	            // Direction error
	            IF #sUDT_HMIStatus.Specific.DirectionErr                                  // Direction verification found the direction fault, stop VSU action and move in opposite direction
	                AND NOT #iqUDT_VSUInterface.MotorRunning                               // The VFD is stopped
	                AND #sx_PEC_EoSFiltered                                                 // The photoeye on the VSU conveyor is empty
	            THEN

	                #sUDT_HMIStatus.Specific.DirectionErr := FALSE;                       // Direction verification found the direction fault, stop VSU action and move in opposite direction

	            END_IF;

	        END_IF;
	    END_REGION

	    REGION 2.2 - Set errors

	        // Exit gap check blocked in movement
	        IF NOT #sx_PEC_GapEnd                                                             // Upper jam sensor occupied
	            AND #iqUDT_VSUInterface.Positioning                                        // The positioning motor is running
	            AND (#sx_UpRequest OR #sx_DownRequest)                                                         // an uprequest is active (going up)
	        THEN

	            #sUDT_HMIStatus.Specific.ExitGapErr := TRUE;                      // Set error upper jam sensor
	        END_IF;

	        // Entry gap check blocked in movement
	        IF NOT #sx_PEC_GapBegin                                                           // Lower jam sensor occupied
	            AND #iqUDT_VSUInterface.Positioning                                        // The positioning motor is running
	            AND (#sx_UpRequest OR #sx_DownRequest)                                                       // an downrequest is active (going down)
	        THEN

	            #sUDT_HMIStatus.Specific.EntryGapErr := TRUE;                      // Set error lower jam sensor
	        END_IF;


	        // Belt tear switch 1
	        IF NOT #ix_BeltTear1                                                   // Belt tear switch 1 is activated
	        THEN
	            #sUDT_HMIStatus.Specific.BeltTear1Err := TRUE;                // set error
	        END_IF;

	        // Belt tear switch 2
	        IF NOT #ix_BeltTear2                                                   // Belt tear switch 2 is activated
	        THEN
	            #sUDT_HMIStatus.Specific.BeltTear2Err := TRUE;                // set error
	        END_IF;

	        // Maintenace supports for lift carriage extracted
	        IF NOT #ix_MaintSupport1                                               // Maintenace support 1 extended
	        THEN
	            #sUDT_HMIStatus.Specific.MaintSupport1Err := TRUE;             // set error
	        END_IF;

	        // Maintenace supports for lift carriage extracted
	        IF NOT #ix_MaintSupport2                                                // Maintenace support 2 extended
	        THEN
	            #sUDT_HMIStatus.Specific.MaintSupport2Err := TRUE;             // set error
	        END_IF;

	        // Upper limit switch
	        IF #ix_LimitSwitchUp                                                   // Upper limit switch is overrun
	        THEN
	            #sUDT_HMIStatus.Specific.UpperPositionErr := TRUE;             // set error
	        END_IF;

	        IF NOT #ix_SafetyDoorDiagUp                                                 // Safety door diagnostic output
	        THEN
	            #sUDT_HMIStatus.Specific.SafetyDoorUpErr := TRUE;                // set error
	        END_IF;


	        // Lower limit switch
	        IF #ix_LimitSwitchDown                                                // Lower limit switch is overrun
	        THEN
	            #sUDT_HMIStatus.Specific.LowerPositionErr := TRUE;            // set error
	        END_IF;

	        IF NOT #ix_SafetyDoorDiagDown                                                 // Safety door diagnostic output
	        THEN
	            #sUDT_HMIStatus.Specific.SafetyDoorDownErr := TRUE;                // set error
	        END_IF;

	        // Direction fault in semiautomatic mode
	        IF #sx_SemiAutomatic                                                               // Running Semi-Automatic
	            AND (((#si_Position = #ci_PositionDown                                     // the requested position is "down"
	            AND #si_DefaultPosition = #ci_PositionDown)                                // and the configured "default" is equal to "down"
	            OR (#si_Position = #ci_PositionDefault                                     // or the request is "default"
	            AND #si_DefaultPosition = #ci_PositionDown)                                // and the configured "default" is equal to "down"
	            AND #sx_DownRequest)                                                       // but the position is "down"

	            OR ((#si_Position = #ci_PositionUp                                         // or the requested position is "up"
	            AND #si_DefaultPosition = #ci_PositionUp)                                  // and the configured "default" is equal to "up"
	            OR (#si_Position = #ci_PositionDefault                                     // or the request is "default"
	            AND #si_DefaultPosition = #ci_PositionUp)                                  // and the configured "default" is equal to "up"
	            AND #sx_UpRequest))                                                        // but the position is "up"
	        THEN

	            #sUDT_HMIStatus.Specific.DirectionErr := TRUE;                            // Direction verification found the Direction fault, stop the parcel
	        END_IF;



	        #sx_ConfigurationError := (#iUDT_VSUConfig.DefaultPosition <= 0);                  // Set the configuration error bit (No status!!)

	    END_REGION

	    REGION 2.3 - Common Error

	        #sUDT_Status.Error :=
	        #iqUDT_VSUInterface.InternalErrorVFD                                           // or there are errors in the VFD
	        OR #iqUDT_VSUInterface.InternalErrorRIOPanel                                   // or an internal error in the RIO panel occured
	        OR #sUDT_HMIStatus.Specific.DirectionErr                                      // Direction verification found the Direction fault, stop the parcel
	        OR #sUDT_HMIStatus.Specific.ExitGapErr                                // Upper jam PEC detected WHILE going Up
	        OR #sUDT_HMIStatus.Specific.EntryGapErr                                // Lower jam PEC detected while going Down
	        OR #sUDT_HMIStatus.Specific.MaintSupport1Err                            // Maintenace carriage support 1 extended in automatic mode
	        OR #sUDT_HMIStatus.Specific.MaintSupport2Err                            // Maintenace carriage support 2 extended in automatic mode
	        OR #sUDT_HMIStatus.Specific.BeltTear1Err                               // Belt tear sensor 1 was detected
	        OR #sUDT_HMIStatus.Specific.BeltTear2Err                              // Belt tear sensor 2 was detected
	        OR #sUDT_HMIStatus.Specific.UpperPositionErr                             // Upper limit switch is overrun
	        OR #sUDT_HMIStatus.Specific.LowerPositionErr                            // Lower limit switch is overrun
	        OR #sUDT_HMIStatus.Specific.SafetyDoorDownErr;                              // Safety door diagnostic fault

	    END_REGION

	    REGION 2.4 - Common Warning

	        // Keyswitch NOT in a position
	        #sUDT_HMIStatus.Specific.KeyswitchWrn := NOT #ix_LCPAutoMode AND NOT #ix_LCPManualMode;
	        #sUDT_Status.Warning := #sUDT_HMIStatus.Specific.KeyswitchWrn;

	    END_REGION

	END_REGION

	REGION 3 - Check conditions to set Equipment ready

	    //Conditions to set bit sx_Ready to operate

	    #sx_Ready := NOT #sUDT_Status.Error                                                // Error present
	    AND #ix_SafetyOk                                                                    // Safety signalling NOT OK
	    AND #iqUDT_VSUInterface.VSUMainPowerOk;                                             // 400v signalling not OK

	    //Enble main contactor
	    #qx_MainContactorOn := (#ix_LCPManualMode OR #ix_LCPAutoMode)                       // Auto or manual enabled
	    AND #ix_OverTempBrakingResistor;                                                    //Temperature breaking resistor is OK


	END_REGION

	REGION 4 - Stop Equipment

	    IF #sx_ManualModeActive                                                             // Manual mode is active
	        AND #sx_AutomaticActive

	        OR (NOT #iqUDT_EquipmentControl.Command.AutomaticOn                            // VSU stops if the bit AutomaticOn from control block is false
	        AND NOT #sx_ManualModeActive)                                                   // Manual mode active bit

	        OR (NOT #sx_Ready                                                               // Bit VSU ready to run in automatic mode
	        AND NOT #sx_ManualModeActive)                                                   // Manual mode active

	        OR NOT #ix_LCPAutoMode                                                          // LCP is not set to automatic
	        OR NOT #ix_SafetyOk                                                             //

	    THEN                                                                                // Order to stop
	        #sx_Stopping := TRUE;                                                           // stopping is activated
	        #sx_AutomaticActive := FALSE;                                                   // switch of automatic activ
	        #sx_StartReceived := FALSE;                                                     // Start command received from system

	    END_IF;

	    IF (#sx_Stopping                                                                     // stopping is activated
	        AND NOT #iqUDT_VSUInterface.Positioning)                                        // The positioning device is not active positioning
	        OR #sFB_MaxStopTime.qx_DelayedSignal
	        OR NOT #sx_Ready

	    THEN
	        #sx_Stopping := FALSE;                                                          // stopping is activated
	        #iqUDT_VSUCommand.CommandUp := FALSE;
	        #iqUDT_VSUCommand.CommandDown := FALSE;
	    END_IF;

	END_REGION

	REGION 5 - Start Automatic mode

	    REGION 5.1 - Start
	        // if start (OS) is received from system, this is memorised until started in cascade
	        IF #iqUDT_EquipmentControl.Command.Start                                       // Start from system
	            AND #sx_Ready                                                               // Equipment has no errors
	        THEN

	            #sx_StartReceived := TRUE;                                                  // Start command received from system

	        END_IF;

	        IF #sx_StartReceived                                                            // Start command received from system
	            AND #iqUDT_VSUInterface.Referenced                                         // and VSU is referenced
	            AND #ix_LCPAutoMode                                                         // and the LCP is set to auto
	        THEN

	            #sx_AutomaticActive := TRUE;                                                // Automatic activated
	            #sx_StartReceived := FALSE;                                                 // Start command received from system
	        END_IF;
	    END_REGION

	    REGION 5.2 - Semi automatic mode

	        #sx_SemiAutomatic := #sx_AutomaticActive                                        // Automatic activated
	        AND #iqUDT_VSUCommand.SemiAutomaticMode;                                       // and Semi-automatic is selected

	    END_REGION

	END_REGION

	REGION 6 - Manual mode

	    REGION 6.1 - Manual mode: activation

	        // Manual mode is active if it is active from hmi or by control block
	        #sx_ManualModeActive := #iqUDT_VSUCommand.ManualMode
	        OR #iqUDT_EquipmentControl.Command.ManualMode
	        OR #ix_LCPManualMode;

	    END_REGION

	    REGION 6.2 - Jog signals

	        #sx_CombinedJogUp :=
	        (((#iqUDT_VSUCommand.ManualMode                                                // HMI in manual
	        OR #iqUDT_EquipmentControl.Command.ManualMode)                                 // Or a system control command to go to manual
	        AND #iqUDT_VSUCommand.JogUp)                                                   // If selected jog in positive direction
	        OR (#ix_LCPManualMode                                                           // box in manual
	        AND #ix_LCPUp));                                                                // If selected jog in positive direction

	        #sx_CombinedJogDown :=
	        (((#iqUDT_VSUCommand.ManualMode                                                 // HMI in manual
	        OR #iqUDT_EquipmentControl.Command.ManualMode)                                  // Or a system control command to go to manual
	        AND #iqUDT_VSUCommand.JogDown)                                                 // If selected jog in negative direction
	        OR (#ix_LCPManualMode                                                           // box in manual
	        AND #ix_LCPDown));                                                              // If selected jog in negative direction

	        // Detecting rising edge on manual jog Up
	        #sR_TRIG_ManualJogUp(CLK := #sx_CombinedJogUp);

	        // Detecting rising edge on manual jog Down
	        #sR_TRIG_ManualJogDown(CLK := #sx_CombinedJogDown);

	    END_REGION

	    REGION 6.3 - Manual mode: disabled

	        // Manual mode bits inputs can be reset in case of malfunction
	        IF #iqUDT_EquipmentControl.Command.DisableManualMode
	        THEN

	            #iqUDT_VSUCommand.ManualMode := FALSE;                                     // reset manual mode
	            #iqUDT_EquipmentControl.Command.ManualMode := FALSE;                       // reset manual mode command
	            #iqUDT_VSUCommand.JogUp := FALSE;                                          // reset manual command Jog Up
	            #iqUDT_VSUCommand.JogDown := FALSE;                                        // reset manual command Jog Down
	            #sx_Jog := FALSE;
	        END_IF;
	    END_REGION

	    REGION 6.4 - Manual PreStart up or down

	        // Pre start conditions to run in manual mode
	        #sx_PreStartManual := #sx_ManualModeActive                                      // Manual mode active bit
	        AND #ix_SafetyOk                                                                // Safety healthy bit
	        //AND #iq_UDT_VSUInterface.PNDeviceOk                                                              // Profinet comunication
	        AND NOT #iqUDT_VSUInterface.InternalErrorVFD;                                  // Internal error from VFD

	        IF #sx_PreStartManual                                                           // Pre start conditions to run in manual mode
	            AND (#sR_TRIG_ManualJogUp.Q                                                  // Trigger to start VSU run in manual jog mode UP
	            OR #sR_TRIG_ManualJogDown.Q)                                                 // Trigger to start VSU run in manual jog mode Down
	            AND NOT #sFB_JogEnable.qx_DelayedSignal
	        THEN

	            #iqUDT_EquipmentControl.Request.SignalingRequest := TRUE;                  // Request signaling TO control block before VSU runs in manual mode

	        END_IF;

	    END_REGION

	    REGION 6.5 - Jog mode Up / Down

	        IF #sx_PreStartManual                                                           // IF in manual jog mode
	            AND (NOT #iqUDT_EquipmentControl.Request.SignalingRequest                  // Signaling request done
	            OR #sFB_JogEnable.qx_DelayedSignal)
	            AND #sx_CombinedJogUp                                                       // If selected jog in positive direction
	            AND NOT #sx_CombinedJogDown                                                 // And not selected jog in negative direction
	        THEN

	            #iqUDT_VSUInterface.JogUp := TRUE;                                         // set jog positive
	            #iqUDT_VSUInterface.JogDown := FALSE;                                      // reset jog negative
	            #sx_Jog := true;

	        ELSIF
	            #sx_PreStartManual                                                          // IF in manual jog mode
	            AND (NOT #iqUDT_EquipmentControl.Request.SignalingRequest                  // Signaling request done
	            OR #sFB_JogEnable.qx_DelayedSignal)
	            AND NOT #sx_CombinedJogUp                                                   // If selected jog in positive direction
	            AND #sx_CombinedJogDown                                                     // and there is command to jog in negative direction
	        THEN

	            #iqUDT_VSUInterface.JogUp := FALSE;                                        // reset jog positive
	            #iqUDT_VSUInterface.JogDown := TRUE;                                       // set jog negative
	            #sx_Jog := true;

	        ELSIF
	            NOT #sx_PreStartManual                                                      // If not in manual mode
	            OR (#sx_PreStartManual                                                      // or in manual mode
	            AND (#sx_CombinedJogUp                                                      // and jog positive is off
	            AND #sx_CombinedJogDown)                                                    // AND jog negative is off
	            OR (NOT #sx_CombinedJogUp                                                   // or jog positive is on
	            AND NOT #sx_CombinedJogDown))                                               // and jog negative is on
	        THEN

	            #iqUDT_VSUInterface.JogUp := FALSE;                                        // reset jog positive
	            #iqUDT_VSUInterface.JogDown := FALSE;                                      // reset jog negative
	            #sx_Jog := False;
	        END_IF;
	    END_REGION
	END_REGION

	REGION 7 - Automatic mode

	    REGION 7.1 - Direction from decision point
	        IF #iqUDT_VSUInterface.RequestedPosition <> 0                                  // Position is received from decision block
	        THEN
	            #si_Position := #iqUDT_VSUInterface.RequestedPosition;                     // Copy the input to the memory

	        END_IF;

	        // Requested position reset
	        IF (#iqUDT_VSUInterface.RequestedPosition = #iqUDT_VSUInterface.PositionActual OR
	            (#iqUDT_VSUInterface.RequestedPosition = #ci_PositionDefault AND #iqUDT_VSUInterface.PositionActual = #si_DefaultPosition))
	        THEN

	            #iqUDT_VSUInterface.RequestedPosition := 0;

	        END_IF;


	    END_REGION

	    REGION 7.2 - Position Up / Down
	        // 2 = Up, 1 = Down and 99 = Default
	        //
	        IF (#si_Position = #ci_PositionUp                                                            // If the position "up" is equal to the request
	            OR (#si_Position = #ci_PositionDefault                                                       // Or the request is "default"
	            AND #si_DefaultPosition = #ci_PositionUp))                                               // and the configured "default" is equal to "up"
	            AND #sx_Ready                                                               // Ready to operate, No errors active
	            AND #sx_AutomaticActive                                                     // Automaticly started
	            AND NOT #sx_SemiAutomatic                                                   // Not running Semi-Automatic
	        THEN

	            #sx_DownRequest := FALSE;                                                   // Reset down command
	            #sx_UpRequest := TRUE;                                                      // Set up command
	            #si_Position := 0;                                                          // Reset the memory
	        END_IF;

	        IF (#si_Position = #ci_PositionDown                                                            // If the position "down" is equal to the request
	            OR (#si_Position = #ci_PositionDefault                                                       // Or the request is "default"
	            AND #si_DefaultPosition = #ci_PositionDown))                                               // and the configured "default" is equal to "down"
	            AND #sx_Ready                                                               // Ready to operate, No errors active
	            AND #sx_AutomaticActive                                                     // Automaticly started
	            AND NOT #sx_SemiAutomatic                                                   // Not running Semi-Automatic
	        THEN

	            #sx_DownRequest := TRUE;                                                    // Set down command
	            #sx_UpRequest := FALSE;                                                     // Reset up command
	            #si_Position := 0;                                                          // Reset the memory
	        END_IF;

	        // if the VSU is not referenced set the default position, this ensures the VSU to go to the default
	        // after refferecing.

	        IF NOT #iqUDT_VSUInterface.Referenced
	        THEN
	            IF #si_DefaultPosition = #ci_PositionUp
	            THEN
	                #sx_DownRequest := FALSE;                                               // Reset down command
	                #sx_UpRequest := TRUE;                                                  // Set up command
	                #iqUDT_VSUInterface.PositionSetpoint := #ci_PositionUp;                             // Set position to be Up
	            END_IF;

	            IF #si_DefaultPosition = #ci_PositionDown
	            THEN
	                #sx_DownRequest := TRUE;                                                // Reset down command
	                #sx_UpRequest := FALSE;                                                 // Set up command
	                #iqUDT_VSUInterface.PositionSetpoint := #ci_PositionDown;                             // Set position to be Down
	            END_IF;
	        END_IF;

	    END_REGION

	    REGION 7.3 - Semi automatic

	        IF #sx_SemiAutomatic                                                            // Not running Semi-Automatic
	            AND #iqUDT_VSUCommand.CommandUp

	        THEN
	            #sx_DownRequest := FALSE;                                                   // Reset down command
	            #sx_UpRequest := TRUE;                                                      // Set up command
	            #iqUDT_VSUCommand.CommandUp := FALSE;
	        END_IF;

	        IF #sx_SemiAutomatic                                                            // Not running Semi-Automatic
	            AND #iqUDT_VSUCommand.CommandDown

	        THEN
	            #sx_DownRequest := TRUE;                                                    // Reset down command
	            #sx_UpRequest := FALSE;                                                     // Set up command
	            #iqUDT_VSUCommand.CommandDown := FALSE;
	        END_IF;

	    END_REGION

	    REGION 7.4 - Controls to to go UP or Down
	        IF #sx_AutomaticActive                                                          // The VSU is automaticly started
	            AND #sx_Ready                                                               // Ready to run / no errors
	        THEN

	            IF #sx_UpRequest                                                            // If there is request to move to the upper position
	                AND #sx_SwitchEnable                                                    // The VSU is enabled to move
	                AND NOT #iqUDT_VSUInterface.Positioning                                // Positioning device is positioning, moving to next position
	                AND #iqUDT_VSUInterface.Ready                                          // the positioning device is errorfree
	                AND NOT #sx_ActualPositionUP                                            // And not in upper position

	            THEN

	                #iqUDT_VSUInterface.PositionSetpoint := #ci_PositionUp;                // Set position to be Up

	            END_IF;

	            IF #sx_DownRequest                                                          // If there is request to move to the lower position
	                AND #sx_SwitchEnable                                                    // The VSU is enabled to move
	                AND NOT #iqUDT_VSUInterface.Positioning                                // Positioning device is positioning, moving to next position
	                AND #iqUDT_VSUInterface.Ready                                          // the positioning device is errorfree
	                AND NOT #sx_ActualPositionDown                                          // And not in lower position

	            THEN

	                #iqUDT_VSUInterface.PositionSetpoint := #ci_PositionDown;              // Set position to be Down

	            END_IF;
	        END_IF;

	    END_REGION

	    REGION 7.5 - Start/Stop VSU conveyor directly
	        // Start
	        IF #iqUDT_EquipmentControl.Command.Start                                       // Start from system
	            AND #sx_Ready                                                               // Equipment has no errors
	        THEN
	            #iqUDT_VSUInterface.ExternalHold := FALSE;                                 // External stop signal
	        END_IF;

	        // Stop
	        IF #sUDT_HMIStatus.Specific.ExitGapErr                                   // Gap check triggered while moving
	            OR #sUDT_HMIStatus.Specific.EntryGapErr                         // Gap check triggered while moving
	            OR #sUDT_HMIStatus.Specific.BeltTear1Err                        // Belt tear detected
	            OR #sUDT_HMIStatus.Specific.BeltTear2Err                        // Belt tear detected
	            OR #sUDT_HMIStatus.Specific.MaintSupport1Err                    // Lift support extracted in automatic mode
	            OR #sUDT_HMIStatus.Specific.MaintSupport2Err                    // Lift support extracted in automatic mode
	            OR #sUDT_HMIStatus.Specific.UpperPositionErr                             // Upper limit switch is overrun
	            OR #sUDT_HMIStatus.Specific.LowerPositionErr                            // Lower limit switch is overrun
	            OR #sUDT_HMIStatus.Specific.SafetyDoorDownErr                               // Safety door diagnostic fault
	            OR #sUDT_HMIStatus.Specific.DirectionErr                                     // in semi-automatic mode and configured as security area: a parcel should go to reject area but direction is not.
	            OR NOT #sx_AutomaticActive                                                  // The VSU is not (semi-)automatic active
	        THEN
	            #iqUDT_VSUInterface.ExternalHold := TRUE;                                  // External stop signal
	        END_IF;
	    END_REGION

	END_REGION

	REGION 8 - Write interface DB signals

	    REGION 8.1 - Signal interface

	        #iqUDT_VSUInterface.InternalErrorReset := #iqUDT_EquipmentControl.Command.Reset;      // Write Reset signal to the VFD interface
	        #iqUDT_VSUInterface.ResetStatistics := #iqUDT_EquipmentControl.Command.ResetData;     // Write Reset data signal to the VFD interface
	        #iqUDT_VSUInterface.SwitchingTime := #iUDT_VSUConfig.SwitchingTime;           // Write switching time from configuration to VFD interface

	    END_REGION

	    REGION 8.2 - Mode selection

	        #iqUDT_VSUInterface.Automatic :=
	        (#sx_AutomaticActive                                                            // Automatic started
	        OR #sx_Stopping                                                                 // stopping is activated
	        OR #sx_PositionAfterRef)                                                        // Go to default position
	        AND #iqUDT_VSUInterface.Referenced;                                            // and the drive is referenced

	        #iqUDT_VSUInterface.Manual :=
	        #sx_ManualModeActive                                                            // Manual mode is started
	        // AND (#sx_CombinedJogUp                                                       // 12.06.24: CombinedJogUp and CombinedJogDown are commented because only manual mode is needed for VFD block
	        // OR #sx_CombinedJogDown)
	        AND #iqUDT_VSUInterface.Referenced;                                            // and the drive is referenced
	    END_REGION

	    REGION 8.3 - Run enable

	        #iqUDT_VSUInterface.RunEnabled :=                                              // Enable the positioning device to run
	        NOT #iqUDT_VSUInterface.InternalErrorVFD                                  // or there are errors in the VFD
	        AND NOT #iqUDT_VSUInterface.InternalErrorRIOPanel                              // or an internal error in the RIO panel occured
	        AND (#iqUDT_VSUInterface.Automatic
	        OR (#iqUDT_VSUInterface.Manual
	        AND (#sx_CombinedJogUp                                                          // If selected jog in positive direction
	        OR #sx_CombinedJogDown))
	        OR #iqUDT_VSUInterface.GoReference);
	    END_REGION

	    REGION 8.4 - Referencing VFD

	        #sR_TRIG_GOReference(CLK := (#sx_AutomaticActive                                 // Refferencing in auto when
	                             AND #sx_StartReceived)                                      // Start command received from system
	                             OR (#sx_ManualModeActive                                    // Manual Refferencing not in auto
	                             AND #iqUDT_VSUCommand.ReferenceRun)                        // Command form HMI to start referecing
	                             OR (#sx_ManualModeActive                                    // Manual Refferencing not in auto
	                             AND #ix_LCPRef));                                           // Command form LCP to start referecing

	        #sR_TRIG_Referenced(CLK := #iqUDT_VSUInterface.Referenced);

	        // Select reference travel and set signalling request prior to VSU movement
	        IF #sR_TRIG_GOReference.Q                                                        // there is rising edge on referencing request bit

	        THEN
	            #iqUDT_VSUInterface.GoReference := TRUE;                                   // Activate the reference travel memory
	            #iqUDT_EquipmentControl.Request.SignalingRequest := TRUE;                  // Request signaling TO control block before running to reference
	        END_IF;

	        // Reference travel mode is active
	        // If signalling request is off set the reference command
	        // if the drive signals to be referenced, reset the command and HMI interface

	        IF #iqUDT_VSUInterface.GoReference = TRUE                                      // The reference travel is activated
	        THEN
	            // 1: Wait for end of signal request to start drive to do its refference run
	            IF NOT #iqUDT_EquipmentControl.Request.SignalingRequest                    // Request signaling TO control block before running to reference
	                AND NOT #sx_PositionAfterRef                                            // last step is active, prohibit starting again.
	            THEN
	                #iqUDT_VSUInterface.Reference_command := TRUE;                         // Reference command, VSU request to do reference run to positioning device

	            END_IF;

	            // 2: Drive did its refference run and is now at refference position
	            IF #sR_TRIG_Referenced.Q                                                     // If the drive is referenced
	            THEN
	                #iqUDT_VSUInterface.Reference_command := FALSE;                        // Reset Reference command, VSU request to do reference run to positioning device
	                #sx_PositionAfterRef := TRUE;                                           // Go to the default position
	                #iqUDT_VSUInterface.PositionActual := 0;
	            END_IF;

	            // 3: go to requested position after which the system can continue
	            IF #iqUDT_VSUInterface.PositionSetpoint = #iqUDT_VSUInterface.PositionActual   // The position is as requested
	                AND #sx_PositionAfterRef

	            THEN
	                #sx_PositionAfterRef := FALSE;                                          // reset to go to the default position
	                #iqUDT_VSUInterface.GoReference := FALSE;                              // Reset the reference travel memory

	            END_IF;
	        END_IF;
	    END_REGION
	END_REGION

	REGION 9 - Statistics

	    // Down Time

	    IF #sx_AutomaticActive                                                              // Automatic active
	        AND NOT #sx_Ready                                                                // Conveyor not ready
	        OR #iqUDT_EquipmentControl.Command.ResetData                                    // Reset statistics
	    THEN

	        "FC_Statistics"(ix_Reset := #iqUDT_EquipmentControl.Command.ResetData,              // Or reset statistics from control
	                        ix_Activate := #sx_AutomaticActive AND NOT #sx_Ready,                // VSU is stopped
	                        ix_RTrigActivate := #sR_TRIG_DownTime.Q,                              // VSU is stopped triger
	                        iqUDT_Statistics := #iqUDT_Statistics.DownTime);                // VSU is stopped statistics
	    END_IF;

	    // Up time

	    IF #sx_AutomaticActive                              // Automatic active
	        AND #sx_Ready                                   // Ready active
	        OR #iqUDT_EquipmentControl.Command.ResetData    // Reset statistics
	    THEN
	        "FC_Statistics"(ix_Reset := #iqUDT_EquipmentControl.Command.ResetData,        // OR reset statistics from control
	                        ix_Activate := #sx_AutomaticActive AND #sx_Ready,                        // VSU is running
	                        ix_RTrigActivate := #sR_TRIG_UpTime.Q,                              // VSU running trigger
	                        iqUDT_Statistics := #iqUDT_Statistics.UpTime);                        // VSU running statistics

	    END_IF;

	    // Exit gap check

	    #sR_TRIG_GapExit_Error(CLK := #sUDT_HMIStatus.Specific.ExitGapErr);               // Oneshot trigger error occurred

	    IF #iqUDT_VSUInterface.ResetStatistics OR                                              // IF there is signal TO reset statistics from VSU interface
	        #iqUDT_EquipmentControl.Command.ResetData OR                                       // Or there is signal to reset statistics from equipment control structure
	        #sUDT_HMIStatus.Specific.ExitGapErr                                        // Or an exit gap check was detected
	    THEN

	        "FC_Statistics"(ix_Reset := #iqUDT_VSUInterface.ResetStatistics OR                 // Reset statistics from HMI
	                        #iqUDT_EquipmentControl.Command.ResetData,                         // Or reset statistics from control
	                        ix_Activate := #sUDT_HMIStatus.Specific.ExitGapErr,        // Upper switch area error occurred
	                        ix_RTrigActivate := #sR_TRIG_GapExit_Error.Q,                          // Error trigger
	                        iqUDT_Statistics := #iqUDT_Statistics.ExitGapErr);          // Statistics of VSU errors

	    END_IF;

	    // Entry gap check

	    #sR_TRIG_GapEntry_Error(CLK := #sUDT_HMIStatus.Specific.EntryGapErr);              // Oneshot trigger error occurred

	    IF #iqUDT_VSUInterface.ResetStatistics OR                                              // IF there is signal TO reset statistics from VSU interface
	        #iqUDT_EquipmentControl.Command.ResetData OR                                       // Or there is signal to reset statistics from equipment control structure
	        #sUDT_HMIStatus.Specific.EntryGapErr                                        // Or an entry gap check was detected
	    THEN

	        "FC_Statistics"(ix_Reset := #iqUDT_VSUInterface.ResetStatistics OR                 // Reset statistics from HMI
	                        #iqUDT_EquipmentControl.Command.ResetData,                         // Or reset statistics from control
	                        ix_Activate := #sUDT_HMIStatus.Specific.EntryGapErr,        // Upper switch area error occurred
	                        ix_RTrigActivate := #sR_TRIG_GapEntry_Error.Q,                         // Error trigger
	                        iqUDT_Statistics := #iqUDT_Statistics.EntryGapErr);          // Statistics of VSU errors

	    END_IF;

	    // Belt tear detection 1

	    #sR_TRIG_BeltTear1(CLK := #sUDT_HMIStatus.Specific.BeltTear1Err);               // Oneshot trigger error occurred

	    IF #iqUDT_VSUInterface.ResetStatistics OR                                              // IF there is signal TO reset statistics from VSU interface
	        #iqUDT_EquipmentControl.Command.ResetData OR                                       // Or there is signal to reset statistics from equipment control structure
	        #sUDT_HMIStatus.Specific.BeltTear1Err                                       // Or an upper switch area error occurred
	    THEN

	        "FC_Statistics"(ix_Reset := #iqUDT_VSUInterface.ResetStatistics OR                 // Reset statistics from HMI
	                        #iqUDT_EquipmentControl.Command.ResetData,                         // Or reset statistics from control
	                        ix_Activate := #sUDT_HMIStatus.Specific.BeltTear1Err,       // Belt tear 1 was detected
	                        ix_RTrigActivate := #sR_TRIG_BeltTear1.Q,                           // Error trigger
	                        iqUDT_Statistics := #iqUDT_Statistics.BeltTear1Err);         // Statistics of VSU errors

	    END_IF;

	    // Belt tear detection 2

	    #sR_TRIG_BeltTear2(CLK := #sUDT_HMIStatus.Specific.BeltTear2Err);              // Oneshot trigger error occurred

	    IF #iqUDT_VSUInterface.ResetStatistics OR                                              // IF there is signal TO reset statistics from VSU interface
	        #iqUDT_EquipmentControl.Command.ResetData OR                                  // Or there is signal to reset statistics from equipment control structure
	        #sUDT_HMIStatus.Specific.BeltTear2Err                                       // Or an upper switch area error occurred
	    THEN

	        "FC_Statistics"(ix_Reset := #iqUDT_VSUInterface.ResetStatistics OR                 // Reset statistics from HMI
	                        #iqUDT_EquipmentControl.Command.ResetData,                         // Or reset statistics from control
	                        ix_Activate := #sUDT_HMIStatus.Specific.BeltTear2Err,         // Belt tear 2 was detected
	                        ix_RTrigActivate := #sR_TRIG_BeltTear2.Q,                          // Error trigger
	                        iqUDT_Statistics := #iqUDT_Statistics.BeltTear2Err);         // Statistics of VSU errors

	    END_IF;

	    // Maintenace support 1 extracted

	    #sR_TRIG_MaintSupport1Err(CLK := #sUDT_HMIStatus.Specific.MaintSupport1Err);              // Oneshot trigger error occurred

	    IF #iqUDT_VSUInterface.ResetStatistics OR                                              // IF there is signal TO reset statistics from VSU interface
	        #iqUDT_EquipmentControl.Command.ResetData OR                                  // Or there is signal to reset statistics from equipment control structure
	        #sUDT_HMIStatus.Specific.MaintSupport1Err                                       // Maintenace support 1 extracted in automatic mode error occurred
	    THEN
	        "FC_Statistics"(ix_Reset := #iqUDT_VSUInterface.ResetStatistics OR                 // Reset statistics from HMI
	                        #iqUDT_EquipmentControl.Command.ResetData,                         // Or reset statistics from control
	                        ix_Activate := #sUDT_HMIStatus.Specific.MaintSupport1Err,         // Maintenace support 1 extracted
	                        ix_RTrigActivate := #sR_TRIG_MaintSupport1Err.Q,                          // Error trigger
	                        iqUDT_Statistics := #iqUDT_Statistics.MaintSupport1Err);         // Statistics of VSU errors
	    END_IF;

	    // Maintenace support 2 extracted

	    #sR_TRIG_MaintSupport2Err(CLK := #sUDT_HMIStatus.Specific.MaintSupport2Err);              // Oneshot trigger error occurred

	    IF #iqUDT_VSUInterface.ResetStatistics OR                                              // IF there is signal TO reset statistics from VSU interface
	        #iqUDT_EquipmentControl.Command.ResetData OR                                  // Or there is signal to reset statistics from equipment control structure
	        #sUDT_HMIStatus.Specific.MaintSupport2Err                                       // Maintenace support 2 extracted in automatic mode error occurred
	    THEN
	        "FC_Statistics"(ix_Reset := #iqUDT_VSUInterface.ResetStatistics OR                 // Reset statistics from HMI
	                        #iqUDT_EquipmentControl.Command.ResetData,                         // Or reset statistics from control
	                        ix_Activate := #sUDT_HMIStatus.Specific.MaintSupport2Err,         // Maintenace support 2 extracted
	                        ix_RTrigActivate := #sR_TRIG_MaintSupport2Err.Q,                          // Error trigger
	                        iqUDT_Statistics := #iqUDT_Statistics.MaintSupport2Err);         // Statistics of VSU errors
	    END_IF;

	    // Limit switch upper position overrun

	    #sR_TRIG_UpperPositionErr(CLK := #sUDT_HMIStatus.Specific.UpperPositionErr);            // Oneshot trigger error occurred

	    IF #iqUDT_VSUInterface.ResetStatistics OR                                              // IF there is signal TO reset statistics from VSU interface
	        #iqUDT_EquipmentControl.Command.ResetData OR                                  // Or there is signal to reset statistics from equipment control structure
	        #sUDT_HMIStatus.Specific.UpperPositionErr                                       // Upper position overrun error occurred
	    THEN
	        "FC_Statistics"(ix_Reset := #iqUDT_VSUInterface.ResetStatistics OR                 // Reset statistics from HMI
	                        #iqUDT_EquipmentControl.Command.ResetData,                         // Or reset statistics from control
	                        ix_Activate := #sUDT_HMIStatus.Specific.UpperPositionErr,         // Limit switch upper position overrun
	                        ix_RTrigActivate := #sR_TRIG_UpperPositionErr.Q,                          // Error trigger
	                        iqUDT_Statistics := #iqUDT_Statistics.UpperPositionErr);         // Statistics of VSU errors
	    END_IF;

	    // Limit switch lower position overrun

	    #sR_TRIG_LowerPositionErr(CLK := #sUDT_HMIStatus.Specific.LowerPositionErr);            // Oneshot trigger error occurred

	    IF #iqUDT_VSUInterface.ResetStatistics OR                                              // IF there is signal TO reset statistics from VSU interface
	        #iqUDT_EquipmentControl.Command.ResetData OR                                  // Or there is signal to reset statistics from equipment control structure
	        #sUDT_HMIStatus.Specific.LowerPositionErr                                       // lower position overrun error occurred
	    THEN
	        "FC_Statistics"(ix_Reset := #iqUDT_VSUInterface.ResetStatistics OR                 // Reset statistics from HMI
	                        #iqUDT_EquipmentControl.Command.ResetData,                         // Or reset statistics from control
	                        ix_Activate := #sUDT_HMIStatus.Specific.LowerPositionErr,         // Limit switch lower position overrun
	                        ix_RTrigActivate := #sR_TRIG_LowerPositionErr.Q,                          // Error trigger
	                        iqUDT_Statistics := #iqUDT_Statistics.LowerPositionErr);         // Statistics of VSU errors
	    END_IF;

	    // Safety door diagnostic fault

	    #sR_TRIG_SafetyDoorErr(CLK := #sUDT_HMIStatus.Specific.SafetyDoorDownErr);

	    IF #iqUDT_VSUInterface.ResetStatistics OR                                              // IF there is signal TO reset statistics from VSU interface
	        #iqUDT_EquipmentControl.Command.ResetData OR                                  // Or there is signal to reset statistics from equipment control structure
	        #sUDT_HMIStatus.Specific.SafetyDoorDownErr                                       // Safety door diagnostic fault
	    THEN
	        "FC_Statistics"(ix_Reset := #iqUDT_VSUInterface.ResetStatistics OR                 // Reset statistics from HMI
	                        #iqUDT_EquipmentControl.Command.ResetData,                         // Or reset statistics from control
	                        ix_Activate := #sUDT_HMIStatus.Specific.SafetyDoorDownErr,         // Safety door diagnostic fault
	                        ix_RTrigActivate := #sR_TRIG_SafetyDoorErr.Q,                          // Error trigger
	                        iqUDT_Statistics := #iqUDT_Statistics.SafetyDoorErr);         // Statistics of VSU errors
	    END_IF;

	    // Direction error

	    #sR_TRIG_Direction_Error(CLK := #sUDT_HMIStatus.Specific.DirectionErr);                 // Oneshot trigger error occurred

	    IF #iqUDT_VSUInterface.ResetStatistics OR                                              // IF there is signal TO reset statistics from VSU interface
	        #iqUDT_EquipmentControl.Command.ResetData OR                                       // Or there is signal to reset statistics from equipment control structure
	        #sUDT_HMIStatus.Specific.DirectionErr                                              // Or an upper switch area error occurred
	    THEN

	        "FC_Statistics"(ix_Reset := #iqUDT_VSUInterface.ResetStatistics OR                 // Reset statistics from HMI
	                        #iqUDT_EquipmentControl.Command.ResetData,                         // Or reset statistics from control
	                        ix_Activate := #sUDT_HMIStatus.Specific.DirectionErr,              // Upper switch area error occurred
	                        ix_RTrigActivate := #sR_TRIG_Direction_Error.Q,                      // Error trigger
	                        iqUDT_Statistics := #iqUDT_Statistics.Direction_Error);                // Statistics of VSU errors

	    END_IF;

	END_REGION

	REGION 10 - Status

	    #sUDT_Status.Stopped := #sx_Ready AND NOT #sx_AutomaticActive AND NOT #sx_Stopping;    // stopped
	    #sUDT_Status.AutoON := #sx_AutomaticActive OR #sx_Stopping;                            // Auto On
	    #sUDT_Status.Halted := FALSE;                                                          // Halted
	    #sUDT_Status.Dieback := FALSE;                                                         // Die back
	    #sUDT_Status.Running := (#sx_UpRequest OR #sx_DownRequest) AND #sx_AutomaticActive;                              // Running
	    #sUDT_Status.ManualRun := #sx_ManualModeActive AND #sUDT_Status.Running;             // Manual run
	    #sUDT_Status.Manual := #sx_ManualModeActive;                                           // Manual
	    #sUDT_Status.EnergySave := FALSE;                                                      // Energy save active
	    #sUDT_Status.SafetyStop := NOT #ix_SafetyOk;                                           // Safety not ok

	    //   Specific status
	    #sUDT_HMIStatus.Specific.ReferencedErr := NOT #iqUDT_VSUInterface.Referenced;
	    #sUDT_HMIStatus.Specific.LiftKeySwitchStop := #ix_LCPStop;
	    #sUDT_HMIStatus.Specific.MaintenanceSwitchUp := #ix_MaintenanceSwitchUp;

	    IF #sUDT_StatusOld <> #sUDT_Status                                            // update on change
	    THEN

	        // Set status to status number
	        #sUDT_HMIStatus.Status := 0;                                               // Initialise status number

	        IF #sUDT_Status.Running                                                    // Running
	        THEN

	            #sUDT_HMIStatus.Status := "DB_HMIStatusConfiguration".Running;

	        END_IF;

	        IF #sUDT_Status.Stopped                                                    // Stopped
	        THEN

	            #sUDT_HMIStatus.Status := "DB_HMIStatusConfiguration".Stopped;

	        END_IF;

	        IF #sUDT_Status.Dieback                                                    // Dieback
	        THEN

	            #sUDT_HMIStatus.Status := "DB_HMIStatusConfiguration".Dieback;

	        END_IF;

	        IF #sUDT_Status.ManualRun                                                  // Manual run
	        THEN

	            #sUDT_HMIStatus.Status := "DB_HMIStatusConfiguration".ManualRun;

	        END_IF;

	        IF #sUDT_Status.Manual                                                     // Manual
	        THEN

	            #sUDT_HMIStatus.Status := "DB_HMIStatusConfiguration".Manual;

	        END_IF;

	        IF #iqUDT_VSUInterface.InternalWarningVFD                                  // The VFD has an internal warning
	            OR #iqUDT_VSUInterface.InternalWarningRIOPanel                         // The RIO panel has an internal warning

	        THEN

	            #sUDT_HMIStatus.Status := "DB_HMIStatusConfiguration".Warning;

	        END_IF;

	        IF #sUDT_HMIStatus.Specific.BeltTear1Err                           // Upper entrance PEC Jam error
	            OR #sUDT_HMIStatus.Specific.BeltTear2Err                       // Lower entrance PEC Jam error
	        THEN

	            #sUDT_HMIStatus.Status := "DB_HMIStatusConfiguration".PECJam;

	        END_IF;

	        IF #sUDT_HMIStatus.Specific.ReferencedErr                                // Refference error
	            OR #sUDT_HMIStatus.Specific.ExitGapErr                        // Upper limit switch error
	            OR #sUDT_HMIStatus.Specific.EntryGapErr                        // Lower limit switch error
	        THEN

	            #sUDT_HMIStatus.Status := "DB_HMIStatusConfiguration".VFDError;

	        END_IF;

	        IF #sUDT_HMIStatus.Specific.DirectionErr                                   // Direction error
	        THEN

	            #sUDT_HMIStatus.Status := "DB_HMIStatusConfiguration".OperationalError;

	        END_IF;


	        IF #sUDT_HMIStatus.Specific.KeyswitchWrn                                  // Key switch error
	            OR #iqUDT_VSUInterface.InternalErrorVFD                                // The VFD has an internal error
	            OR #iqUDT_VSUInterface.InternalErrorRIOPanel                           // The RIO panel has an internal error
	        THEN

	            #sUDT_HMIStatus.Status := "DB_HMIStatusConfiguration".Error;

	        END_IF;


	        IF #sUDT_Status.SafetyStop                                                 // Safety stop
	        THEN

	            #sUDT_HMIStatus.Status := "DB_HMIStatusConfiguration".SafetyStop;

	        END_IF;

	        #qUDT_HMIStatus := #sUDT_HMIStatus;                                       // Copy status to output
	        #sUDT_StatusOld := #sUDT_Status;                                          // Copy status TO memory
	        #qUDT_Status := #sUDT_Status;                                             // Copy status to output
	    END_IF;

	    #qUDT_HMIStatus.Specific.UpperPositionErr := #sx_ActualPositionUP;
	    #qUDT_HMIStatus.Specific.LowerPositionErr := #sx_ActualPositionDown;

	END_REGION

	REGION 11 - Report to control block

	    "FC_EquipmentReport"(iUDT_Status := #sUDT_Status,
	                         iqUDT_Control := #iqUDT_EquipmentControl);

	END_REGION
END_FUNCTION_BLOCK

TYPE "UDT_WSRBufferState"
VERSION : 0.1
   STRUCT
      Destination : Int;
      BufferState1 : Struct
         BinRequest : Bool;
         BinSend : Bool;
         UpcomingBarcode : String[30];
         WaintingTime : Int;
      END_STRUCT;
      BufferState2 : Struct
         BinRequest : Bool;
         BinSend : Bool;
         UpcomingBarcode : String[30];
         WaintingTime : Int;
      END_STRUCT;
      BufferState3 : Struct
         BinRequest : Bool;
         BinSend : Bool;
         UpcomingBarcode : String[30];
         WaintingTime : Int;
      END_STRUCT;
   END_STRUCT;

END_TYPE

TYPE "UDT_WSRCommonStatus"
VERSION : 0.1
   STRUCT
      "010" { S7_SetPoint := 'False'} : "UDT_CommonStatus";
      "020" { S7_SetPoint := 'False'} : "UDT_CommonStatus";
      "030" { S7_SetPoint := 'False'} : "UDT_CommonStatus";
      "040" { S7_SetPoint := 'False'} : "UDT_CommonStatus";
      "041" { S7_SetPoint := 'False'} : "UDT_CommonStatus";
      "050" { S7_SetPoint := 'False'} : "UDT_CommonStatus";
      "060" { S7_SetPoint := 'False'} : "UDT_CommonStatus";
      "070" { S7_SetPoint := 'False'} : "UDT_CommonStatus";
      "080" { S7_SetPoint := 'False'} : "UDT_CommonStatus";
      "110" { S7_SetPoint := 'False'} : "UDT_CommonStatus";
      "120" { S7_SetPoint := 'False'} : "UDT_CommonStatus";
      "130" { S7_SetPoint := 'False'} : "UDT_CommonStatus";
      "140" { S7_SetPoint := 'False'} : "UDT_CommonStatus";
      "141" { S7_SetPoint := 'False'} : "UDT_CommonStatus";
      "150" { S7_SetPoint := 'False'} : "UDT_CommonStatus";
      "160" { S7_SetPoint := 'False'} : "UDT_CommonStatus";
      "170" { S7_SetPoint := 'False'} : "UDT_CommonStatus";
      "180" { S7_SetPoint := 'False'} : "UDT_CommonStatus";
      "210" { S7_SetPoint := 'False'} : "UDT_CommonStatus";
      "220" { S7_SetPoint := 'False'} : "UDT_CommonStatus";
      "230" { S7_SetPoint := 'False'} : "UDT_CommonStatus";
      "240" { S7_SetPoint := 'False'} : "UDT_CommonStatus";
      "241" { S7_SetPoint := 'False'} : "UDT_CommonStatus";
      "250" { S7_SetPoint := 'False'} : "UDT_CommonStatus";
      "260" { S7_SetPoint := 'False'} : "UDT_CommonStatus";
      "270" { S7_SetPoint := 'False'} : "UDT_CommonStatus";
   END_STRUCT;

END_TYPE

TYPE "UDT_WSRStatus"
VERSION : 0.1
   STRUCT
      "010" { S7_SetPoint := 'False'} : "UDT_StatusTC03";
      "020" { S7_SetPoint := 'False'} : "UDT_StatusTC13";
      "030" { S7_SetPoint := 'False'} : "UDT_StatusTC03";
      "040" { S7_SetPoint := 'False'} : "UDT_StatusTC07";
      "041" { S7_SetPoint := 'False'} : "UDT_StatusTC36";
      "050" { S7_SetPoint := 'False'} : "UDT_StatusTC03";
      "060" { S7_SetPoint := 'False'} : "UDT_StatusTC13";
      "070" { S7_SetPoint := 'False'} : "UDT_StatusTC03";
      "080" { S7_SetPoint := 'False'} : "UDT_StatusTC13";
      "110" { S7_SetPoint := 'False'} : "UDT_StatusTC03";
      "120" { S7_SetPoint := 'False'} : "UDT_StatusTC13";
      "130" { S7_SetPoint := 'False'} : "UDT_StatusTC03";
      "140" { S7_SetPoint := 'False'} : "UDT_StatusTC07";
      "141" { S7_SetPoint := 'False'} : "UDT_StatusTC36";
      "150" { S7_SetPoint := 'False'} : "UDT_StatusTC03";
      "160" { S7_SetPoint := 'False'} : "UDT_StatusTC13";
      "170" { S7_SetPoint := 'False'} : "UDT_StatusTC03";
      "180" { S7_SetPoint := 'False'} : "UDT_StatusTC12";
      "210" { S7_SetPoint := 'False'} : "UDT_StatusTC03";
      "220" { S7_SetPoint := 'False'} : "UDT_StatusTC13";
      "230" { S7_SetPoint := 'False'} : "UDT_StatusTC03";
      "240" { S7_SetPoint := 'False'} : "UDT_StatusTC02";
      "241" { S7_SetPoint := 'False'} : "UDT_StatusTC36";
      "250" { S7_SetPoint := 'False'} : "UDT_StatusTC03";
      "260" { S7_SetPoint := 'False'} : "UDT_StatusTC13";
      "270" { S7_SetPoint := 'False'} : "UDT_StatusTC03";
   END_STRUCT;

END_TYPE

TYPE "UDT_WSRConfiguration"
VERSION : 0.1
   STRUCT
      GlobalConfig : Struct
         LeftStationAvailable : Bool := TRUE;
         RightStationAvailable : Bool := TRUE;
         OperationTimeout : UDInt;
         DestinationEmpty : Int;
         DestinationPartialy : Int;
         GINRangeStart : Int;
         GINRangeEnd : Int;
         BinReleaseDistance : Int;
         BinOrderTimeout : Int;
      END_STRUCT;
      "010" : Struct
         Conveyor { S7_SetPoint := 'False'} : "UDT_ConveyorConfiguration";
         PEC_EoS : "UDT_PECUpdateConfiguration";
         MCO_M01 : "UDT_AixPlcFullControllerConfiguration";
      END_STRUCT;
      "020" : Struct
         Conveyor { S7_SetPoint := 'False'} : "UDT_ConveyorConfiguration";
         PEC_EoS : "UDT_PECUpdateConfiguration";
         MCO_M01 : "UDT_AixPlcFullControllerConfiguration";
      END_STRUCT;
      "030" : Struct
         Conveyor { S7_SetPoint := 'False'} : "UDT_ConveyorConfiguration";
         PEC_EoS : "UDT_PECUpdateConfiguration";
         MCO_M01 : "UDT_AixPlcFullControllerConfiguration";
      END_STRUCT;
      "040" : Struct
         Conveyor { S7_SetPoint := 'False'} : "UDT_ConveyorConfiguration";
         PEC_EoS : "UDT_PECConfiguration";
         MCO_M01 : "UDT_AixPlcFullControllerConfiguration";
         BladeStopEoS : "UDT_ValveConfiguration";
      END_STRUCT;
      "041" : Struct
         Conveyor { S7_SetPoint := 'False'} : "UDT_ConveyorConfiguration";
         RightAngledTransfer : "UDT_RATConfiguration";
         MCO_M01 : "UDT_AixPlcFullControllerConfiguration";
      END_STRUCT;
      "050" : Struct
         Conveyor { S7_SetPoint := 'False'} : "UDT_ConveyorConfiguration";
         PEC_EoS : "UDT_PECUpdateConfiguration";
         MCO_M01 : "UDT_AixPlcFullControllerConfiguration";
      END_STRUCT;
      "060" : Struct
         Conveyor { S7_SetPoint := 'False'} : "UDT_ConveyorConfiguration";
         PEC_EoS : "UDT_PECUpdateConfiguration";
         MCO_M01 : "UDT_AixPlcFullControllerConfiguration";
      END_STRUCT;
      "070" : Struct
         Conveyor { S7_SetPoint := 'False'} : "UDT_ConveyorConfiguration";
         PEC_EoS : "UDT_PECUpdateConfiguration";
         MCO_M01 : "UDT_AixPlcFullControllerConfiguration";
      END_STRUCT;
      "080" : Struct
         Conveyor { S7_SetPoint := 'False'} : "UDT_ConveyorConfiguration";
         PEC_EoS : "UDT_PECUpdateConfiguration";
         MCO_M01 : "UDT_AixPlcFullControllerConfiguration";
      END_STRUCT;
      "110" : Struct
         Conveyor { S7_SetPoint := 'False'} : "UDT_ConveyorConfiguration";
         PEC_EoS : "UDT_PECUpdateConfiguration";
         MCO_M01 : "UDT_AixPlcFullControllerConfiguration";
      END_STRUCT;
      "120" : Struct
         Conveyor { S7_SetPoint := 'False'} : "UDT_ConveyorConfiguration";
         PEC_EoS : "UDT_PECUpdateConfiguration";
         MCO_M01 : "UDT_AixPlcFullControllerConfiguration";
      END_STRUCT;
      "130" : Struct
         Conveyor { S7_SetPoint := 'False'} : "UDT_ConveyorConfiguration";
         PEC_EoS : "UDT_PECUpdateConfiguration";
         MCO_M01 : "UDT_AixPlcFullControllerConfiguration";
      END_STRUCT;
      "140" : Struct
         Conveyor { S7_SetPoint := 'False'} : "UDT_ConveyorConfiguration";
         PEC_EoS : "UDT_PECConfiguration";
         MCO_M01 : "UDT_AixPlcFullControllerConfiguration";
         BladeStopEoS : "UDT_ValveConfiguration";
      END_STRUCT;
      "141" : Struct
         Conveyor { S7_SetPoint := 'False'} : "UDT_ConveyorConfiguration";
         RightAngledTransfer : "UDT_RATConfiguration";
         MCO_M01 : "UDT_AixPlcFullControllerConfiguration";
      END_STRUCT;
      "150" : Struct
         Conveyor { S7_SetPoint := 'False'} : "UDT_ConveyorConfiguration";
         PEC_EoS : "UDT_PECUpdateConfiguration";
         MCO_M01 : "UDT_AixPlcFullControllerConfiguration";
      END_STRUCT;
      "160" : Struct
         Conveyor { S7_SetPoint := 'False'} : "UDT_ConveyorConfiguration";
         PEC_EoS : "UDT_PECUpdateConfiguration";
         MCO_M01 : "UDT_AixPlcFullControllerConfiguration";
      END_STRUCT;
      "170" : Struct
         Conveyor { S7_SetPoint := 'False'} : "UDT_ConveyorConfiguration";
         PEC_EoS : "UDT_PECUpdateConfiguration";
         MCO_M01 : "UDT_AixPlcFullControllerConfiguration";
      END_STRUCT;
      "180" : Struct
         Conveyor { S7_SetPoint := 'False'} : "UDT_ConveyorConfiguration";
         PEC_EoS : "UDT_PECConfiguration";
         MCO_M01 : "UDT_AixPlcFullControllerConfiguration";
      END_STRUCT;
      "210" : Struct
         Conveyor { S7_SetPoint := 'False'} : "UDT_ConveyorConfiguration";
         PEC_EoS : "UDT_PECUpdateConfiguration";
         MCO_M01 : "UDT_AixPlcFullControllerConfiguration";
      END_STRUCT;
      "220" : Struct
         Conveyor { S7_SetPoint := 'False'} : "UDT_ConveyorConfiguration";
         PEC_EoS : "UDT_PECUpdateConfiguration";
         MCO_M01 : "UDT_AixPlcFullControllerConfiguration";
      END_STRUCT;
      "230" : Struct
         Conveyor { S7_SetPoint := 'False'} : "UDT_ConveyorConfiguration";
         PEC_EoS : "UDT_PECUpdateConfiguration";
         MCO_M01 : "UDT_AixPlcFullControllerConfiguration";
      END_STRUCT;
      "240" : Struct
         Conveyor { S7_SetPoint := 'False'} : "UDT_ConveyorConfiguration";
         PEC_EoS : "UDT_PECConfiguration";
         MCO_M01 : "UDT_AixPlcFullControllerConfiguration";
      END_STRUCT;
      "241" : Struct
         Conveyor { S7_SetPoint := 'False'} : "UDT_ConveyorConfiguration";
         RightAngledTransfer : "UDT_RATConfiguration";
         MCO_M01 : "UDT_AixPlcFullControllerConfiguration";
      END_STRUCT;
      "250" : Struct
         Conveyor { S7_SetPoint := 'False'} : "UDT_ConveyorConfiguration";
         PEC_EoS : "UDT_PECUpdateConfiguration";
         MCO_M01 : "UDT_AixPlcFullControllerConfiguration";
      END_STRUCT;
      "260" : Struct
         Conveyor { S7_SetPoint := 'False'} : "UDT_ConveyorConfiguration";
         PEC_EoS : "UDT_PECUpdateConfiguration";
         MCO_M01 : "UDT_AixPlcFullControllerConfiguration";
      END_STRUCT;
      "270" : Struct
         Conveyor { S7_SetPoint := 'False'} : "UDT_ConveyorConfiguration";
         PEC_EoS : "UDT_PECUpdateConfiguration";
         MCO_M01 : "UDT_AixPlcFullControllerConfiguration";
      END_STRUCT;
   END_STRUCT;

END_TYPE

TYPE "UDT_CrossoverCommand"
VERSION : 0.1
   STRUCT
      ManualMode : Bool;   // Manual mode command from HMI
      ManualUp : Bool;   // Command to move devise up
      ManualDown : Bool;   // Command to move devise down
   END_STRUCT;

END_TYPE

TYPE "UDT_WSRHmiCommands"
VERSION : 0.1
   STRUCT
      "010" { S7_SetPoint := 'False'} : "UDT_HMICommandTCxx";
      "020" { S7_SetPoint := 'False'} : "UDT_HMICommandTCxx";
      "030" { S7_SetPoint := 'False'} : "UDT_HMICommandTCxx";
      "040" { S7_SetPoint := 'False'} : "UDT_HMICommandTC07";
      "041" : "UDT_HMICommandTC36";
      "050" : "UDT_HMICommandTCxx";
      "060" { S7_SetPoint := 'False'} : "UDT_HMICommandTCxx";
      "070" { S7_SetPoint := 'False'} : "UDT_HMICommandTCxx";
      "080" { S7_SetPoint := 'False'} : "UDT_HMICommandTCxx";
      "110" { S7_SetPoint := 'False'} : "UDT_HMICommandTCxx";
      "120" { S7_SetPoint := 'False'} : "UDT_HMICommandTCxx";
      "130" { S7_SetPoint := 'False'} : "UDT_HMICommandTCxx";
      "140" { S7_SetPoint := 'False'} : "UDT_HMICommandTC07";
      "141" : "UDT_HMICommandTC36";
      "150" { S7_SetPoint := 'False'} : "UDT_HMICommandTCxx";
      "160" { S7_SetPoint := 'False'} : "UDT_HMICommandTCxx";
      "170" { S7_SetPoint := 'False'} : "UDT_HMICommandTCxx";
      "180" { S7_SetPoint := 'False'} : "UDT_HMICommandTCxx";
      "210" { S7_SetPoint := 'False'} : "UDT_HMICommandTCxx";
      "220" { S7_SetPoint := 'False'} : "UDT_HMICommandTCxx";
      "230" { S7_SetPoint := 'False'} : "UDT_HMICommandTCxx";
      "240" { S7_SetPoint := 'False'} : "UDT_HMICommandTCxx";
      "241" : "UDT_HMICommandTC36";
      "250" { S7_SetPoint := 'False'} : "UDT_HMICommandTCxx";
      "260" { S7_SetPoint := 'False'} : "UDT_HMICommandTCxx";
      "270" { S7_SetPoint := 'False'} : "UDT_HMICommandTCxx";
   END_STRUCT;

END_TYPE

FUNCTION_BLOCK "FB_Tracking"
TITLE = FB_Tracking
{ S7_Optimized_Access := 'TRUE' }
AUTHOR : MHSE
FAMILY : GeneralSystemFunctions
VERSION : 3.0
// ATTRIBUTES
// AUTO_NUMBER = True
// BLOCK_NUMBER = 33
// END_ATTRIBUTES
//Function block to shift data in the tracking array.
   VAR_INPUT
      iUDT_ConveyorCommonConfiguration { ExternalAccessible := 'False'; ExternalVisible := 'False'; ExternalWritable := 'False'} : "UDT_ConveyorCommonConfiguration";   // Conveyor common configuration
   END_VAR

   VAR_IN_OUT
      iqa_TrackingData : Array[*] of Int;   // Tracking array
      iqUDT_ConveyorInterface : "UDT_ConveyorInterface";   // Conveyor interface
      iqUDT_HandshakeUp : "UDT_ConveyorHandshake";   // Upstream conveyor handshake
      iqUDT_Handshake : "UDT_ConveyorHandshake";   // Conveyor handshake
   END_VAR

   VAR
      si_TrackingArrayLen { ExternalAccessible := 'False'; ExternalVisible := 'False'; ExternalWritable := 'False'} : Int;   // Tracking array length
      si_TrackingArrayLowBound { ExternalAccessible := 'False'; ExternalVisible := 'False'; ExternalWritable := 'False'} : Int;   // Tracking array lower bound
      sdi_TotalConvLength { ExternalAccessible := 'False'; ExternalVisible := 'False'; ExternalWritable := 'False'} : DInt;   // Number of tracking entries is equal to the conveyor length in cm
      si_Displacement { ExternalAccessible := 'False'; ExternalVisible := 'False'; ExternalWritable := 'False'} : Int;   // Displacement
      si_ShiftDestination { ExternalAccessible := 'False'; ExternalVisible := 'False'; ExternalWritable := 'False'} : Int;   // Pointer to the entry to start writing the tracking data
      si_ShiftOffset { ExternalAccessible := 'False'; ExternalVisible := 'False'; ExternalWritable := 'False'} : Int;   // Number of entries to be shifted and its direction
      sdi_GINInsertPosition { ExternalAccessible := 'False'; ExternalVisible := 'False'; ExternalWritable := 'False'} : DInt;   // Position where GIN form upstream conveyor will be inserted
      sdi_GINExtractPosition { ExternalAccessible := 'False'; ExternalVisible := 'False'; ExternalWritable := 'False'} : DInt;   // Position from which GIN will be moved to the downstream conveyor
      sx_InvalidTrackArraySize { ExternalAccessible := 'False'; ExternalVisible := 'False'; ExternalWritable := 'False'} : Bool;   // Invalid tracking array size
   END_VAR


BEGIN
	(*
	----------------------------------------------------------------------------------------
	|                                                                                      |
	|  Copyright  2019             MHS                                                     |
	|  All Rights Reserved         Larenweg 90                                             |
	|                              5234 KC 's-Hertogenbosch,                               |
	|                              Netherlands                                             |
	|                                                                                      |
	----------------------------------------------------------------------------------------

	Version history:
	Date        | Version   | Author       | Remark
	----------------------------------------------------------------------------------------
	24/05/2019  | 0.1       | L. Klar      | first release MHS TIA 15.1
	14/06/2019  | 0.2       | A.Nowak      | Replacement of instruction if for direct write into variable - Region 3
	19/07/2019  | 0.5       | L.Klar       | Status handling changed
	24/07/2019  | 2.0       | L.Klar       | 2.0 MHS library release TIA 15.1
	23/08/2019  | 2.1       | L.Klar       | "UDT_ConveyorConfiguration" changed to "UDT_ConveyorCommonConfiguration", internal tracking error set instead of coil assigment.
	10/09/2019  | 2.2       | L.Klar       | Comments changed, block optimized
	21/10/2019  | 2.3       | L.Klar       | Configuration UDT chanaged to input
	12/11/2019  | 3.0       | P.Majka      | 3.0 MHS library release TIA 15.1
	20/12/2019  | 3.1       | S. Deulkar   | Used configureation error bit to report to conveyor block
	15/01/2020  | 3.2       | L.Klar       | Block adjusted to allow to transfer negative GIN numbers
	*)

	REGION 1 – Get the required number of entries

	    // Number of entries is a conveyor length in cm
	    #sdi_TotalConvLength := (#iUDT_ConveyorCommonConfiguration.Length + #iUDT_ConveyorCommonConfiguration.LengthCorrection) / 10;

	END_REGION

	REGION 2 – Number of tracking records validation

	    // Tracking array dimensions
	    #si_TrackingArrayLen := "FC_GetNrOfArrayEl"(#iqa_TrackingData);
	    #si_TrackingArrayLowBound := DINT_TO_INT(LOWER_BOUND(ARR := #iqa_TrackingData, DIM := 1));

	    // Check if the number of entries is exceeding the tracking array size
	    #sx_InvalidTrackArraySize := #si_TrackingArrayLen < #sdi_TotalConvLength + 2
	    OR #si_TrackingArrayLowBound <> 0;

	END_REGION

	REGION 3 – Read the displacement

	    #si_Displacement := #iqUDT_ConveyorInterface.Displacement;

	END_REGION

	REGION 4 – Prepare tracking array pointers

	    // A conveyor can run in forward and reverse direction
	    // Data will be shifted into tracking entry position 1 for both cases.
	    #si_ShiftDestination := 1;

	    // If the direction is forward (positive displacement), entry 2 is taken as offset (shifts conveyor length from pos 2 in pos 1)
	    IF #si_Displacement > 0
	    THEN

	        #si_ShiftOffset := 2;
	        #sdi_GINInsertPosition := #sdi_TotalConvLength + 1;
	        #sdi_GINExtractPosition := 1;

	        // If the direction is reverse (negative displacement), entry 0 is taken as offset (shifts conveyor length from pos 0 in pos 1)
	    ELSE

	        #si_ShiftOffset := 0;
	        #sdi_GINInsertPosition := 0;
	        #sdi_GINExtractPosition := #sdi_TotalConvLength;

	    END_IF;

	END_REGION

	REGION 5 – Shift data

	    // Data is shifted only if the conveyor is running (positive or negtive displacement)
	    WHILE #si_Displacement <> 0 DO

	        // Conveyor running forward
	        IF (#si_Displacement > 0)
	        THEN

	            // GIN is moved into the tracking array on GIN insert position if the number of positions in upstream conveyor handshake is available
	            // The number of positions to be shifted will be decremented
	            IF (#iqUDT_HandshakeUp.GIN <> 0
	                AND #iqUDT_HandshakeUp.NrOfPosToShift > 0)
	            THEN

	                #iqa_TrackingData[#sdi_GINInsertPosition] := #iqUDT_HandshakeUp.GIN;
	                #iqUDT_HandshakeUp.NrOfPosToShift -= 1;

	            ELSIF (#iqUDT_HandshakeUp.GIN <> 0
	                AND #iqUDT_HandshakeUp.NrOfPosToShift = 0)
	            THEN

	                #iqa_TrackingData[#sdi_GINInsertPosition] := #iqUDT_HandshakeUp.GIN;

	            END_IF;

	            // Clear the downsteam handshake GIN if the number of positions to be shifted is 0
	            IF (#iqUDT_Handshake.GIN <> 0 AND #iqUDT_Handshake.NrOfPosToShift = 0)
	            THEN

	                #iqUDT_Handshake.GIN := 0;

	            END_IF;

	            // GIN is moved into the handshake structure if the data is available at GIN extract position
	            // The number of positions will be incremented
	            IF (#iqa_TrackingData[#sdi_GINExtractPosition] <> 0)
	            THEN

	                IF (#iqUDT_Handshake.GIN = 0)
	                THEN

	                    #iqUDT_Handshake.GIN := #iqa_TrackingData[#sdi_GINExtractPosition];
	                    #iqUDT_Handshake.NrOfPosToShift += 1;

	                ELSIF (#iqUDT_Handshake.GIN = #iqa_TrackingData[#sdi_GINExtractPosition])
	                THEN

	                    #iqUDT_Handshake.NrOfPosToShift += 1;

	                END_IF;

	            END_IF;

	            // Update displacement
	            #si_Displacement -= 1;

	            // Conveyor running backward
	        ELSIF (#si_Displacement < 0)
	        THEN

	            // GIN is moved into the tracking array on GIN insert position if the number of positions in downstream conveyor handshake is available
	            // The number of positions to be shifted will be decremented
	            IF (#iqUDT_Handshake.GIN <> 0
	                AND #iqUDT_Handshake.NrOfPosToShift > 0)
	            THEN

	                #iqa_TrackingData[#sdi_GINInsertPosition] := #iqUDT_Handshake.GIN;
	                #iqUDT_Handshake.NrOfPosToShift -= 1;

	                // In case of displacement greater than 1 and no positions to be shifted the GIN will be written to avoid gaps in data
	                // Writing will be stopped when GIN 0 is detected
	            ELSIF (#iqUDT_Handshake.GIN <> 0
	                AND #iqUDT_Handshake.NrOfPosToShift = 0)
	            THEN

	                #iqa_TrackingData[#sdi_GINInsertPosition] := #iqUDT_Handshake.GIN;

	            END_IF;

	            // Clear the upstream handshake GIN if the number of positions to be shifted is 0
	            IF (#iqUDT_HandshakeUp.GIN <> 0 AND #iqUDT_HandshakeUp.NrOfPosToShift = 0)
	            THEN

	                #iqUDT_HandshakeUp.GIN := 0;

	            END_IF;

	            // GIN is moved into the handshake structure if the data is available at GIN extract position
	            // The number of positions will be incremented
	            IF (#iqa_TrackingData[#sdi_GINExtractPosition] <> 0)
	            THEN

	                IF (#iqUDT_HandshakeUp.GIN = 0)
	                THEN

	                    #iqUDT_HandshakeUp.GIN := #iqa_TrackingData[#sdi_GINExtractPosition];
	                    #iqUDT_HandshakeUp.NrOfPosToShift += 1;

	                    // In case of displacement greater than 1 and no positions to be shifted the GIN will be written to avoid gaps in data
	                    // Writing will be stopped when GIN 0 is detected
	                ELSIF (#iqUDT_HandshakeUp.GIN = #iqa_TrackingData[#sdi_GINExtractPosition])
	                THEN

	                    #iqUDT_HandshakeUp.NrOfPosToShift += 1;

	                END_IF;

	            END_IF;

	            // Update displacement
	            #si_Displacement += 1;

	        END_IF;

	        // Shift the total conveyor length (number of tracking array entries) one cm up or down
	        MOVE_BLK(IN := #iqa_TrackingData[#si_ShiftOffset],
	                 COUNT := DINT_TO_ULINT(#sdi_TotalConvLength),
	                 OUT => #iqa_TrackingData[#si_ShiftDestination]);

	        // Clear the GIN insert position
	        #iqa_TrackingData[#sdi_GINInsertPosition] := 0;

	    END_WHILE;

	END_REGION

	REGION 6 – Internal tracking error

	    // The internal tracking error is set to stop the conveyor
	    // It is reset in the conveyor block
	    IF (#sx_InvalidTrackArraySize)
	    THEN

	        #iqUDT_ConveyorInterface.ConfigurationError := TRUE;

	    END_IF;

	END_REGION
END_FUNCTION_BLOCK

FUNCTION_BLOCK "FB_MCOConveyLinxAixController"
TITLE = FB_VfdConveyLinxAixController
{ S7_Optimized_Access := 'TRUE' }
AUTHOR : Fortna
VERSION : 4.0
//Function to interface with ConveyLinx Aix Controller. On the controller is the possibility to connect two motors with two photoeyes and run the motors independent from each other. Also can each motor output used as a "normal" on/off output
//--V4.0 split the function to accomodate only 1 Motor
   VAR_INPUT
      iUDT_AixConfig { ExternalAccessible := 'False'; ExternalVisible := 'False'; ExternalWritable := 'False'} : "UDT_AixPlcFullControllerConfiguration";   // Configuration structure
      iUDT_AixInputsModule { ExternalAccessible := 'False'; ExternalVisible := 'False'; ExternalWritable := 'False'} : "UDT_AixPlcFullIn";   // ConveyLinxAix inputs structure
      ii_MotorPositionId { ExternalAccessible := 'False'; ExternalVisible := 'False'; ExternalWritable := 'False'} : Int;   // 1 = Master Left, 2 = Master Right, 11 Slave Left, 12 Slave Right
      ii_PositionSetpoint { ExternalAccessible := 'False'; ExternalVisible := 'False'; ExternalWritable := 'False'} : Int;
      ix_24vOk { ExternalAccessible := 'False'; ExternalVisible := 'False'; ExternalWritable := 'False'} : Bool;   // TRUE when 24VDC is healthy
      ix_SimulationModeActive { ExternalAccessible := 'False'; ExternalVisible := 'False'; ExternalWritable := 'False'} : Bool;   // TRUE when Simulation mode active
      ix_StartPositioning { ExternalAccessible := 'False'; ExternalVisible := 'False'; ExternalWritable := 'False'} : Bool;
      ix_ResetPosition { ExternalAccessible := 'False'; ExternalVisible := 'False'; ExternalWritable := 'False'} : Bool;
   END_VAR

   VAR_OUTPUT
      qUDT_HMIStatus { ExternalAccessible := 'False'; ExternalVisible := 'False'; ExternalWritable := 'False'} : "UDT_AixControllerStatus";   // HMI status structure for right motor
      qx_Positioned { ExternalAccessible := 'False'; ExternalVisible := 'False'; ExternalWritable := 'False'} : Bool;
   END_VAR

   VAR_IN_OUT
      iqUDT_AixOutputsModule : "UDT_AixPlcFullOut";   // ConveyLinxAix nr.1 outputs structure
      iqUDT_ConveyorInterface : "UDT_ConveyorInterface";   // Conveyor interface structure Motor
      iqUDT_MCOStatistics : "UDT_VfdStatistics";   // Satistics structure
   END_VAR

   VAR
      sFB_TimerOnOffDelayMCOSpeedFeedbackError { ExternalAccessible := 'False'; ExternalVisible := 'False'; ExternalWritable := 'False'; S7_SetPoint := 'False'} : "FB_TimerOnOffDelay";
      sFB_TimerOnOffDelayCheck24V { ExternalAccessible := 'False'; ExternalVisible := 'False'; ExternalWritable := 'False'; S7_SetPoint := 'False'} : "FB_TimerOnOffDelay";   // MHS "TimerOnOffDelay" - to delay time for MCO 24V contactor
      sFB_TimerOnOffDelayMCO { ExternalAccessible := 'False'; ExternalVisible := 'False'; ExternalWritable := 'False'; S7_SetPoint := 'False'} : "FB_TimerOnOffDelay";
      sFB_TimerOnOffDelayMCOReset { ExternalAccessible := 'False'; ExternalVisible := 'False'; ExternalWritable := 'False'; S7_SetPoint := 'False'} : "FB_TimerOnOffDelay";   // MHS "TimerOnOffDelay" - to extend MCO reset
      sFB_TimerOnOffDelayMCORunningFeedbackError { ExternalAccessible := 'False'; ExternalVisible := 'False'; ExternalWritable := 'False'; S7_SetPoint := 'False'} : "FB_TimerOnOffDelay";
      sFB_TimerOnOffDelayAcceleration { ExternalAccessible := 'False'; ExternalVisible := 'False'; ExternalWritable := 'False'; S7_SetPoint := 'False'} : "FB_TimerOnOffDelay";
      sUDT_HMIStatus { ExternalAccessible := 'False'; ExternalVisible := 'False'; ExternalWritable := 'False'; S7_SetPoint := 'False'} : "UDT_AixControllerStatus";   // Detailed MCO status overview
      sUDT_PNDeviceController { ExternalAccessible := 'False'; ExternalVisible := 'False'; ExternalWritable := 'False'; S7_SetPoint := 'False'} : "UDT_PNDevice";   // PN device info structure, Controller 1
      ss_PNPortsStatusController { ExternalAccessible := 'False'; ExternalVisible := 'False'; ExternalWritable := 'False'} : Array[1..8] of Bool;   // TRUE when specific port has an error, Controller
      sR_TRIG_PNSlaveNotOnline {InstructionName := 'R_TRIG'; LibVersion := '1.0'; ExternalAccessible := 'False'; ExternalVisible := 'False'; ExternalWritable := 'False'; S7_SetPoint := 'False'} : R_TRIG;   // Rising edge for trigger Profinet slave not online statistics
      sR_TRIG_PNSlaveError {InstructionName := 'R_TRIG'; LibVersion := '1.0'; ExternalAccessible := 'False'; ExternalVisible := 'False'; ExternalWritable := 'False'; S7_SetPoint := 'False'} : R_TRIG;   // Rising edge for trigger Profinet slave error statistics
      sR_TRIG_MCOInternalError {InstructionName := 'R_TRIG'; LibVersion := '1.0'; ExternalAccessible := 'False'; ExternalVisible := 'False'; ExternalWritable := 'False'; S7_SetPoint := 'False'} : R_TRIG;   // Rising edge for trigger Internal MCO Error statistics
      sR_TRIG_Running {InstructionName := 'R_TRIG'; LibVersion := '1.0'; ExternalAccessible := 'False'; ExternalVisible := 'False'; ExternalWritable := 'False'; S7_SetPoint := 'False'} : R_TRIG;   // Rising edge for trigger running motor
      sR_TRIG_CommunicationErrorMCO {InstructionName := 'R_TRIG'; LibVersion := '1.0'; ExternalAccessible := 'False'; ExternalVisible := 'False'; ExternalWritable := 'False'; S7_SetPoint := 'False'} : R_TRIG;   // Rising edge for trigger communication error
      sR_TRIG_ResetPosition {InstructionName := 'R_TRIG'; LibVersion := '1.0'; ExternalAccessible := 'False'; ExternalVisible := 'False'; ExternalWritable := 'False'; S7_SetPoint := 'False'} : R_TRIG;   // Rising edge reset position
      sF_TRIG_RunFwd {InstructionName := 'F_TRIG'; LibVersion := '1.0'; ExternalAccessible := 'False'; ExternalVisible := 'False'; ExternalWritable := 'False'; S7_SetPoint := 'False'} : F_TRIG;   // Falling edge for run forward signal
      sF_TRIG_RunRvs {InstructionName := 'F_TRIG'; LibVersion := '1.0'; ExternalAccessible := 'False'; ExternalVisible := 'False'; ExternalWritable := 'False'; S7_SetPoint := 'False'} : F_TRIG;   // Falling edge for run reverse signal
      sr_ActualSpeedSetpoint { ExternalAccessible := 'False'; ExternalVisible := 'False'; ExternalWritable := 'False'} : Real;   // Actual speed setpoint motor
      si_ActualSpeed { ExternalAccessible := 'False'; ExternalVisible := 'False'; ExternalWritable := 'False'} : Int;   // Actual speed motor
      si_MotorAcceleration { ExternalAccessible := 'False'; ExternalVisible := 'False'; ExternalWritable := 'False'} : Int;   // Left motor acceleration
      si_MotorDeceleration { ExternalAccessible := 'False'; ExternalVisible := 'False'; ExternalWritable := 'False'} : Int;   // Motor deceleration
      si_LeftMotorPosition { ExternalAccessible := 'False'; ExternalVisible := 'False'; ExternalWritable := 'False'} : Int;   // Left motor actual position
      si_LastLeftMotorPosition { ExternalAccessible := 'False'; ExternalVisible := 'False'; ExternalWritable := 'False'} : Int;   // Left motor last cycle position
      si_RightMotorPosition { ExternalAccessible := 'False'; ExternalVisible := 'False'; ExternalWritable := 'False'} : Int;   // Right motor actual position
      si_LastRightMotorPosition { ExternalAccessible := 'False'; ExternalVisible := 'False'; ExternalWritable := 'False'} : Int;   // Right motor last cycle position
      sx_GeneralStatisticsReset { ExternalAccessible := 'False'; ExternalVisible := 'False'; ExternalWritable := 'False'} : Bool;   // Reset from or right conveyor
      sx_HardwareOK { ExternalAccessible := 'False'; ExternalVisible := 'False'; ExternalWritable := 'False'} : Bool;   // Hardware is ok
      sx_ConfigurationError { ExternalAccessible := 'False'; ExternalVisible := 'False'; ExternalWritable := 'False'} : Bool;   // Commissioning: configuration error
      sx_PNDeviceHealthyControler { ExternalAccessible := 'False'; ExternalVisible := 'False'; ExternalWritable := 'False'} : Bool;   // Profinet device is online and error free, Controller 1
      sx_AixAvailableControler { ExternalAccessible := 'False'; ExternalVisible := 'False'; ExternalWritable := 'False'} : Bool;   // Hardware of MCO is ok and no communication error with movikit, Controller 1
      sx_24vOk { ExternalAccessible := 'False'; ExternalVisible := 'False'; ExternalWritable := 'False'} : Bool;   // 24VDC is healthy
      sx_ErrorActive { ExternalAccessible := 'False'; ExternalVisible := 'False'; ExternalWritable := 'False'} : Bool;   // Block has an error
      sx_EnableOperation { ExternalAccessible := 'False'; ExternalVisible := 'False'; ExternalWritable := 'False'} : Bool;   // Enable operation signal
      sx_RunForward { ExternalAccessible := 'False'; ExternalVisible := 'False'; ExternalWritable := 'False'} : Bool;   // Start MCO forward
      sx_RunReverse { ExternalAccessible := 'False'; ExternalVisible := 'False'; ExternalWritable := 'False'} : Bool;   // Start MCO backward
      sx_SpeedSetpointReached { ExternalAccessible := 'False'; ExternalVisible := 'False'; ExternalWritable := 'False'} : Bool;   // Speed setpoint reached motor
      sx_SpeedFeedbackError { ExternalAccessible := 'False'; ExternalVisible := 'False'; ExternalWritable := 'False'} : Bool;   // motor speed feedback error
      sx_ErrorController { ExternalAccessible := 'False'; ExternalVisible := 'False'; ExternalWritable := 'False'} : Bool;   // Active if any erorr from controller 1 is active
      sx_ErrorCMotor { ExternalAccessible := 'False'; ExternalVisible := 'False'; ExternalWritable := 'False'} : Bool;   // TRUE if error from controler motor is active
      sx_Accelerating { ExternalAccessible := 'False'; ExternalVisible := 'False'; ExternalWritable := 'False'} : Bool;   // Motor acceleration
      sx_HardwareOk_Motor { ExternalAccessible := 'False'; ExternalVisible := 'False'; ExternalWritable := 'False'} : Bool;   // Motor hardware ok
      sx_LeftServoHomeHasBeenSet { ExternalAccessible := 'False'; ExternalVisible := 'False'; ExternalWritable := 'False'} : Bool;   // Servo position has beeen reset to 0
      sx_RightServoHomeHasBeenSet { ExternalAccessible := 'False'; ExternalVisible := 'False'; ExternalWritable := 'False'} : Bool;   // Servo position has beeen reset to 0
      sb_MotorRotationStatus { ExternalAccessible := 'False'; ExternalVisible := 'False'; ExternalWritable := 'False'} : Byte;   // 0 Motor not running, Normal or Servo Braking Mode applied; 1 Motor running in CCW Direction; 2 Motor running in CW Direction; 3 Motor not running and Free Braking Mode applied
   END_VAR

   VAR CONSTANT
      ci_MCOArea : UInt := 1;   // Area ID of IO Profinet devices
      ci_SubmoduleHWType : UInt := 5;   // Submodule HW_type number
      ci_TelegramSlot : UInt := 1;   // Free Siemens telegram slot
      ci_TelegramSubslot : UInt := 3;   // Free Siemens telegram subslot
      ci_NumberOfProfinetPorts : Int := 2;   // Number of Profinet ports in device
      cr_MaximumOutput : Real := 16384.0;   // PLC maximum output value
      cw_ActualSpeedMask : Word := 2#0011_1111_1111_1111;   // Mask to get the speed from the profinet MotorActualSpeed Word
      cudi_ExtendedResetTime : UDInt := 500;   // Extending the reset puls
      cudi_HardwareCheckDelay : UDInt := 2000;   // Delay to enable hardware to start up, checking will start after this time
      cudi_FeedbackErrorDelay : UDInt := 10000;   // Maximum delaytime deviation from setpoint is allowed
      cudi_TimeOffsetSpeedmonitoring : UDInt := 2000;   // Additional time
      cudi_HeartbeatDelay : UDInt := 5000;   // Maximum dely between heartbeat
      ci_Master_Left : Int := 1;
      ci_Master_Right : Int := 2;
      ci_Slave_Left : Int := 11;
      ci_Slave_Right : Int := 12;
   END_VAR


BEGIN
	(*
	----------------------------------------------------------------------------------------

	Version history:
	Date        | Version   | Author        | Remark
	----------------------------------------------------------------------------------------
	03/01/2022  | 1.0       | N.Kadam       | First release MHSE TIA 16.0
	24/03/2022  | 1.1       | M.Piela       | Bug fix, adding running feedback error
	05/05/2022  | 1.2       | M.Piela       | Status update
	31/05/2022  | 1.3       | M.Piela       | Ramp up/down calculation fix
	21/07/2022  | 1.4       | M.Piela       | Prevent motor to go below the minimum speed
	29/07/2022  | 1.5       | M.Piela       | Status update, add hardware ok to the profinet checking
	01/08/2022  | 1.6       | M.Piela       | Add Hardware ok to reset internal error
	01/08/2022  | 1.7       | G.Vlooswijk   | Fix to make it possible to run 1 of the 2 motors
	                                        | Check setpoint instead of sx_EnableOperation for Feedback Error check
	                                        | Removed if statement i_UDT_Ai2Config.DirectionReversal, speed from controller always positive
	06/08/2022  | 1.8       | G.Vlooswijk   | Removed minimal speedsetpoint
	05/07/2023  | 1.9       | F.Baten       | Complete separation of 2 motors
	13/09/2023  | 4.0       | F.Baten       | Reorganised structure and took out unused symbolics
	                                        | Status as 1 controller with 2 seperate controlled motors
	02/05/2024  | 5.0       | I.Ajram       | Split the function to accomodate only 1 Motor, added an input to indicate which motor to control
	08/05/2024  | 5.1       | S.Nieswiec    | qUDT_AixOutputsModule move to in/out variables, name changed to iqUDT_AixOutputsModule
	08/05/2024  | 5.2       | K. Pokorski   | Add displacement calculation
	13/05/2024  | 5.3       | K. Pokorski   | Add roller ratio
	08/06/2024  | 5.4       | S.Nieswiec    | Fixed servo delta calculation (went back to previous functioning version), adjusted region numbering
	                                        | displacement was negative on some conveyors while positive on others
	21/06/2024  | 5.5       | I.Ajram       | Added Master / Slave Mod, Slave is used when one conveyor is controlling more than 1 MCO, the rest will act/ be configured as slaves
	*)

	REGION 1 - Get Device Profinet information

	    //Get Device Profinet name, Controller
	    "FC_GetDevicePN"(is_PNDeviceName := #iUDT_AixConfig.AixContrlPNDeviceName,
	                     ix_SimulationModeActive := #ix_SimulationModeActive,
	                     iqUDT_PND := #sUDT_PNDeviceController);

	    //Get number of ports, Controller
	    "FC_GetPNPortStatus"(ii_NumberOfPorts := #ci_NumberOfProfinetPorts,
	                         iUDT_DevicePNInfo := #sUDT_PNDeviceController,
	                         qa_PortFault => #ss_PNPortsStatusController);

	END_REGION

	REGION 2 - Reset errors


	    REGION 2.1 - Motor

	        // Reset errors when InternalErrorReset is given
	        IF #iqUDT_ConveyorInterface.InternalErrorReset OR (NOT #iqUDT_ConveyorInterface.HardwareOk AND #sUDT_HMIStatus.PNSlaveNotOnline)
	        THEN
	            #sUDT_HMIStatus.PNSlaveNotOnline := FALSE;
	            #sUDT_HMIStatus.PNSlaveError := FALSE;
	            #sUDT_HMIStatus.InternalError := FALSE;
	            #sUDT_HMIStatus.PNSlaveWarning := FALSE;
	            #sUDT_HMIStatus.SpeedFeedbackError := FALSE;
	            #sx_SpeedFeedbackError := FALSE;
	            #sx_ErrorCMotor := FALSE;
	            #sUDT_HMIStatus.MotorStatus.Overheat := FALSE;
	            #sUDT_HMIStatus.MotorStatus.MaxTorque := FALSE;
	            #sUDT_HMIStatus.MotorStatus.ShortCircuit := FALSE;
	            #sUDT_HMIStatus.MotorStatus.MotorNotConnected := FALSE;
	            #sUDT_HMIStatus.MotorStatus.Overload := FALSE;
	            #sUDT_HMIStatus.MotorStatus.Stalled := FALSE;
	            #sUDT_HMIStatus.MotorStatus.BadHall := FALSE;
	            #sUDT_HMIStatus.MotorStatus.BoardOverheat := FALSE;
	            #sUDT_HMIStatus.MotorStatus.OverVoltage := FALSE;
	            #sUDT_HMIStatus.MotorStatus.LowVoltage := FALSE;
	            #iqUDT_ConveyorInterface.InternalErrorVFD := FALSE;

	        END_IF;

	    END_REGION

	    REGION 2.2 - Reset pulse
	        // Create extended pulse for MCO Reset
	        #sFB_TimerOnOffDelayMCOReset(iudi_OnDelayTime := #cudi_ExtendedResetTime,
	                                     iudi_OffDelayTime := 0,
	                                     ix_SignalToDelay := #iqUDT_AixOutputsModule.ClearMotorError = 1,
	                                     ix_Enable := TRUE);
	        // set the reset signal directly when reset is active
	        IF #iqUDT_ConveyorInterface.InternalErrorReset THEN
	            #iqUDT_AixOutputsModule.ClearMotorError := 1;
	        END_IF;

	        // Reset the ClearMotorError after 500[ms] pulse
	        IF #sFB_TimerOnOffDelayMCOReset.qx_DelayedSignal
	        THEN
	            #iqUDT_AixOutputsModule.ClearMotorError := 0;
	        END_IF;

	    END_REGION

	END_REGION

	REGION 3 - Hardware checks

	    // Hardware will only be available after the delay, so the device has time for the initialisation
	    #sFB_TimerOnOffDelayCheck24V(iudi_OnDelayTime := #cudi_HardwareCheckDelay,
	                                 ix_SignalToDelay := #ix_24vOk);

	    #sx_24vOk := #sFB_TimerOnOffDelayCheck24V.qx_DelayedSignal;

	    #sx_HardwareOk_Motor := #iqUDT_ConveyorInterface.HardwareOk AND #iUDT_AixConfig.Motor.MotorExist;

	    #sx_HardwareOK := NOT #ix_SimulationModeActive
	    AND #sx_24vOk
	    AND (#sx_HardwareOk_Motor OR NOT #iUDT_AixConfig.Motor.MotorExist)
	    AND (#ss_PNPortsStatusController[1] OR #ss_PNPortsStatusController[2])
	    AND #iqUDT_ConveyorInterface.HardwareOk;


	    // Check if PN device is online
	    IF NOT "DB_ProfinetDiagnostic".ProfinetNetworks[#sUDT_PNDeviceController.PNNetworknumber].DeviceStatus[#sUDT_PNDeviceController.PNDeviceNumber].DeviceState.Exist
	        AND #sx_HardwareOK
	    THEN
	        #sUDT_HMIStatus.PNSlaveNotOnline := TRUE;
	    END_IF;

	    // Check IF PN ports are healthy
	    IF #ss_PNPortsStatusController[1] XOR #ss_PNPortsStatusController[2]

	    THEN
	        #sUDT_HMIStatus.PNSlaveWarning := TRUE;
	    END_IF;

	    // Check if PN device has an error
	    IF "DB_ProfinetDiagnostic".ProfinetNetworks[#sUDT_PNDeviceController.PNNetworknumber].DeviceStatus[#sUDT_PNDeviceController.PNDeviceNumber].DeviceState.Error
	        AND #sx_HardwareOK
	        AND NOT #sUDT_HMIStatus.PNSlaveWarning
	    THEN
	        #sUDT_HMIStatus.PNSlaveError := TRUE;
	    END_IF;

	    // Set bit when PN device is healthy (online and no error)
	    #sx_PNDeviceHealthyControler := NOT #sUDT_HMIStatus.PNSlaveNotOnline
	    AND NOT #sUDT_HMIStatus.PNSlaveError
	    AND #sUDT_PNDeviceController.PNDeviceFound
	    AND #sx_24vOk;

	    // Set hardware available bit when all conditions are met
	    #sx_AixAvailableControler := (#sx_24vOk
	    AND #sx_PNDeviceHealthyControler
	    AND (#sx_HardwareOk_Motor OR NOT #iUDT_AixConfig.Motor.MotorExist))
	    OR #ix_SimulationModeActive;

	    // Check communication (heartbeat)
	    #sFB_TimerOnOffDelayMCO(iudi_OnDelayTime := #cudi_HeartbeatDelay,
	                            ix_SignalToDelay := NOT #iUDT_AixInputsModule.AllSensorPortInputs.Heartbeat);

	    // Set error when MoviKit communication is not available
	    IF #sFB_TimerOnOffDelayMCO.qx_DelayedSignal AND #sx_HardwareOK
	    THEN

	        #sUDT_HMIStatus.CommunicationErrorVFD := TRUE;

	    END_IF;
	END_REGION

	REGION 4 - Check errors and warnings
	    REGION 4.1 - Error from controller for right motor
	        IF #ii_MotorPositionId = #ci_Master_Right OR #ii_MotorPositionId = #ci_Slave_Right THEN
	            //Write errors to UDT_Status
	            IF #iUDT_AixInputsModule.RightMotorDiagnostic.Overheat
	            THEN
	                #sUDT_HMIStatus.MotorStatus.Overheat := TRUE;
	            END_IF;

	            #sUDT_HMIStatus.MotorStatus.MaxTorque := #iUDT_AixInputsModule.RightMotorDiagnostic.MaxTorque;

	            IF #iUDT_AixInputsModule.RightMotorDiagnostic.ShortCircuit
	            THEN
	                #sUDT_HMIStatus.MotorStatus.ShortCircuit := TRUE;
	            END_IF;

	            IF #iUDT_AixInputsModule.RightMotorDiagnostic.MotorNotConnected
	            THEN
	                #sUDT_HMIStatus.MotorStatus.MotorNotConnected := TRUE;
	            END_IF;

	            IF #iUDT_AixInputsModule.RightMotorDiagnostic.Overload
	            THEN
	                #sUDT_HMIStatus.MotorStatus.Overload := TRUE;
	            END_IF;

	            IF #iUDT_AixInputsModule.RightMotorDiagnostic.Stalled
	            THEN
	                #sUDT_HMIStatus.MotorStatus.Stalled := TRUE;
	            END_IF;

	            IF #iUDT_AixInputsModule.RightMotorDiagnostic.BadHall
	            THEN
	                #sUDT_HMIStatus.MotorStatus.BadHall := TRUE;
	            END_IF;

	            IF #iUDT_AixInputsModule.RightMotorDiagnostic.BoardOverheat
	            THEN
	                #sUDT_HMIStatus.MotorStatus.BoardOverheat := TRUE;
	            END_IF;

	            IF #iUDT_AixInputsModule.RightMotorDiagnostic.OverVoltage
	            THEN
	                #sUDT_HMIStatus.MotorStatus.OverVoltage := TRUE;
	            END_IF;

	            IF #iUDT_AixInputsModule.RightMotorDiagnostic.LowVoltage
	            THEN
	                #sUDT_HMIStatus.MotorStatus.LowVoltage := TRUE;
	            END_IF;

	        END_IF;
	    END_REGION

	    REGION 4.2 - Error from controller for left motor
	        IF #ii_MotorPositionId = #ci_Master_Left OR #ii_MotorPositionId = #ci_Slave_Left THEN
	            //Write errors to UDT_Status
	            IF #iUDT_AixInputsModule.LeftMotorDiagnostic.Overheat
	            THEN
	                #sUDT_HMIStatus.MotorStatus.Overheat := TRUE;
	            END_IF;

	            #sUDT_HMIStatus.MotorStatus.MaxTorque := #iUDT_AixInputsModule.LeftMotorDiagnostic.MaxTorque;

	            IF #iUDT_AixInputsModule.LeftMotorDiagnostic.ShortCircuit
	            THEN
	                #sUDT_HMIStatus.MotorStatus.ShortCircuit := TRUE;
	            END_IF;

	            IF #iUDT_AixInputsModule.LeftMotorDiagnostic.MotorNotConnected
	            THEN
	                #sUDT_HMIStatus.MotorStatus.MotorNotConnected := TRUE;
	            END_IF;

	            IF #iUDT_AixInputsModule.LeftMotorDiagnostic.Overload
	            THEN
	                #sUDT_HMIStatus.MotorStatus.Overload := TRUE;
	            END_IF;

	            IF #iUDT_AixInputsModule.LeftMotorDiagnostic.Stalled
	            THEN
	                #sUDT_HMIStatus.MotorStatus.Stalled := TRUE;
	            END_IF;

	            IF #iUDT_AixInputsModule.LeftMotorDiagnostic.BadHall
	            THEN
	                #sUDT_HMIStatus.MotorStatus.BadHall := TRUE;
	            END_IF;

	            IF #iUDT_AixInputsModule.LeftMotorDiagnostic.BoardOverheat
	            THEN
	                #sUDT_HMIStatus.MotorStatus.BoardOverheat := TRUE;
	            END_IF;

	            IF #iUDT_AixInputsModule.LeftMotorDiagnostic.OverVoltage
	            THEN
	                #sUDT_HMIStatus.MotorStatus.OverVoltage := TRUE;
	            END_IF;

	            IF #iUDT_AixInputsModule.LeftMotorDiagnostic.LowVoltage
	            THEN
	                #sUDT_HMIStatus.MotorStatus.LowVoltage := TRUE;
	            END_IF;
	        END_IF;
	    END_REGION

	    REGION 4.3 - Collective Error
	        //If any error from controller motor ocursed then set error to TRUE
	        IF #iUDT_AixConfig.Motor.MotorExist
	        THEN
	            #sx_ErrorCMotor := #sUDT_HMIStatus.MotorStatus.Overheat OR
	            // #sUDT_HMIStatus.MotorError.MaxTorque OR
	            #sUDT_HMIStatus.MotorStatus.ShortCircuit OR
	            #sUDT_HMIStatus.MotorStatus.MotorNotConnected OR
	            #sUDT_HMIStatus.MotorStatus.Overload OR
	            #sUDT_HMIStatus.MotorStatus.Stalled OR
	            #sUDT_HMIStatus.MotorStatus.BadHall OR
	            #sUDT_HMIStatus.MotorStatus.BoardOverheat OR
	            #sUDT_HMIStatus.MotorStatus.OverVoltage OR
	            #sUDT_HMIStatus.MotorStatus.LowVoltage OR
	            #sUDT_HMIStatus.SpeedFeedbackError OR
	            #sUDT_HMIStatus.PNSlaveNotOnline OR
	            #sUDT_HMIStatus.PNSlaveError;
	        END_IF;
	    END_REGION

	    REGION 4.4 - Controller general

	        // Error Controller is two drives combined
	        #sx_ErrorController :=
	        #iUDT_AixInputsModule.ConveyStopStatus.StopActiveLostConn OR
	        #iUDT_AixInputsModule.ConveyStopStatus.StopActiveLostPLC OR
	        #sx_ErrorCMotor OR
	        FALSE;

